SUBAPPLICATION Seitenschieber (* Subapplication Type *)
  (* Standard: 61499-2 *)
  (* Version 1.0, 2023-01-29, Franz *)
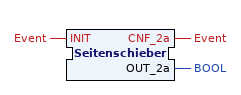
  EVENT_INPUT
    INIT;
  END_EVENT
  EVENT_OUTPUT
    CNF_2a;
  END_EVENT
  VAR_OUTPUT
    OUT_2a : BOOL;
  END_VAR
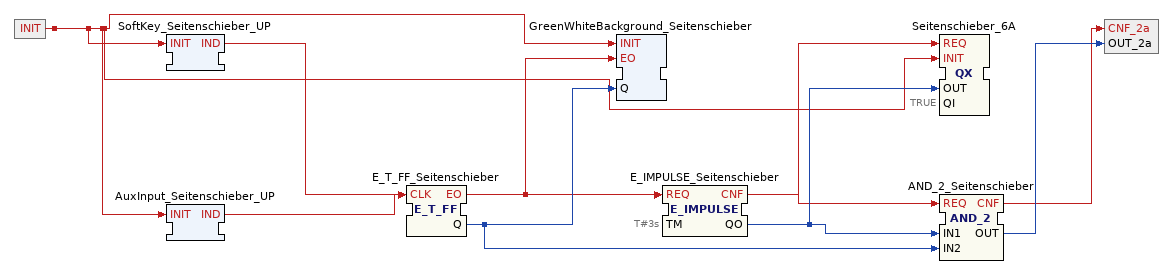
  FBS
    AND_2_Seitenschieber : AND_2;
    E_T_FF_Seitenschieber : E_T_FF;
    Seitenschieber_6A : QX(QI := TRUE);
    E_IMPULSE_Seitenschieber : E_IMPULSE(TM := T#3s);
  END_FBS
  SUBAPPLICATION AuxInput_Seitenschieber_UP
    EVENT_INPUT
      INIT;
    END_EVENT
    EVENT_OUTPUT
      IND;
    END_EVENT
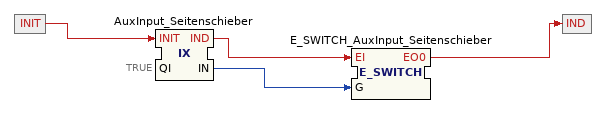
    FBS
      E_SWITCH_AuxInput_Seitenschieber : E_SWITCH;
      AuxInput_Seitenschieber : IX(QI := TRUE);
    END_FBS
    EVENT_CONNECTIONS
      AuxInput_Seitenschieber.IND TO E_SWITCH_AuxInput_Seitenschieber.EI;
      INIT TO AuxInput_Seitenschieber.INIT;
      E_SWITCH_AuxInput_Seitenschieber.EO0 TO IND;
    END_CONNECTIONS
    DATA_CONNECTIONS
      AuxInput_Seitenschieber.IN TO E_SWITCH_AuxInput_Seitenschieber.G;
    END_CONNECTIONS
  END_SUBAPPLICATION
  SUBAPPLICATION SoftKey_Seitenschieber_UP
    EVENT_INPUT
      INIT;
    END_EVENT
    EVENT_OUTPUT
      IND;
    END_EVENT
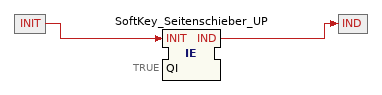
    FBS
      SoftKey_Seitenschieber_UP : IE(QI := TRUE);
    END_FBS
    EVENT_CONNECTIONS
      INIT TO SoftKey_Seitenschieber_UP.INIT;
      SoftKey_Seitenschieber_UP.IND TO IND;
    END_CONNECTIONS
  END_SUBAPPLICATION
  SUBAPPLICATION GreenWhiteBackground_Seitenschieber
    EVENT_INPUT
      INIT;
      EO;
    END_EVENT
    VAR_INPUT
      Q : BOOL;
    END_VAR
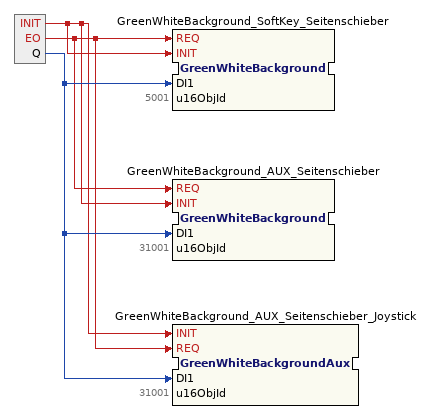
    FBS
      GreenWhiteBackground_SoftKey_Seitenschieber : GreenWhiteBackground(u16ObjId := 5001);
      GreenWhiteBackground_AUX_Seitenschieber : GreenWhiteBackground(u16ObjId := 31001);
      GreenWhiteBackground_AUX_Seitenschieber_Joystick : GreenWhiteBackgroundAux(u16ObjId := 31001);
    END_FBS
    EVENT_CONNECTIONS
      EO TO GreenWhiteBackground_SoftKey_Seitenschieber.REQ;
      INIT TO GreenWhiteBackground_SoftKey_Seitenschieber.INIT;
      EO TO GreenWhiteBackground_AUX_Seitenschieber.REQ;
      INIT TO GreenWhiteBackground_AUX_Seitenschieber.INIT;
      INIT TO GreenWhiteBackground_AUX_Seitenschieber_Joystick.INIT;
      EO TO GreenWhiteBackground_AUX_Seitenschieber_Joystick.REQ;
    END_CONNECTIONS
    DATA_CONNECTIONS
      Q TO GreenWhiteBackground_SoftKey_Seitenschieber.DI1;
      Q TO GreenWhiteBackground_AUX_Seitenschieber.DI1;
      Q TO GreenWhiteBackground_AUX_Seitenschieber_Joystick.DI1;
    END_CONNECTIONS
  END_SUBAPPLICATION
  EVENT_CONNECTIONS
    E_IMPULSE_Seitenschieber.CNF TO AND_2_Seitenschieber.REQ;
    E_T_FF_Seitenschieber.EO TO E_IMPULSE_Seitenschieber.REQ;
    E_IMPULSE_Seitenschieber.CNF TO Seitenschieber_6A.REQ;
    AND_2_Seitenschieber.CNF TO CNF_2a;
    INIT TO SoftKey_Seitenschieber_UP.INIT;
    SoftKey_Seitenschieber_UP.IND TO E_T_FF_Seitenschieber.CLK;
    INIT TO AuxInput_Seitenschieber_UP.INIT;
    AuxInput_Seitenschieber_UP.IND TO E_T_FF_Seitenschieber.CLK;
    INIT TO Seitenschieber_6A.INIT;
    INIT TO GreenWhiteBackground_Seitenschieber.INIT;
    E_T_FF_Seitenschieber.EO TO GreenWhiteBackground_Seitenschieber.EO;
  END_CONNECTIONS
  DATA_CONNECTIONS
    E_IMPULSE_Seitenschieber.QO TO AND_2_Seitenschieber.IN1;
    E_T_FF_Seitenschieber.Q TO AND_2_Seitenschieber.IN2;
    E_IMPULSE_Seitenschieber.QO TO Seitenschieber_6A.OUT;
    AND_2_Seitenschieber.OUT TO OUT_2a;
    E_T_FF_Seitenschieber.Q TO GreenWhiteBackground_Seitenschieber.Q;
  END_CONNECTIONS
END_SUBAPPLICATION
